TYPE McWriteParameterArgs :
STRUCT
	///Number of the parameter
	parameterNumber: INT;
	///Value to write
	value: LREAL;
END_STRUCT
END_TYPE

(* stored: Version 1.1.0.1, ProductVersion 3.1.4019.2
   DUT McWriteParameterArgs: Id {e706e5f1-566b-4413-bce6-c06f56ef9d4c} *)
